DATA_BLOCK "PilzData"
VAR
  "85A1" : STRUCT
    I8 : Bool;
    I9 : Bool;
    I10 : Bool;
    I11 : Bool;
    I12 : Bool;
    I13 : Bool;
    I14 : Bool;
    I15 : Bool;
    I0 : Bool;
    I1 : Bool;
    I2 : Bool;
    I3 : Bool;
    I4 : Bool;
    I5 : Bool;
    I6 : Bool;
    I7 : Bool;
    I24 : Bool;
    I25 : Bool;
    I26 : Bool;
    I27 : Bool;
    I28 : Bool;
    I29 : Bool;
    I30 : Bool;
    I31 : Bool;
    I16 : Bool;
    I17 : Bool;
    I18 : Bool;
    I19 : Bool;
    I20 : Bool;
    I21 : Bool;
    I22 : Bool;
    I23 : Bool;
    O0 : Bool;
    O1 : Bool;
    O2 : Bool;
    O3 : Bool;
    Spare_1 : Bool;
    Spare_2 : Bool;
    Spare_3 : Bool;
    Spare_4 : Bool;
    Spare_5 : Bool;
    Spare_6 : Bool;
    Spare_7 : Bool;
    Spare_8 : Bool;
    Spare_9 : Bool;
    Spare_10 : Bool;
    Spare_11 : Bool;
    Spare_12 : Bool;
  END_STRUCT;
  "85A2" : STRUCT
    I0 : Bool;
    I1 : Bool;
    I2 : Bool;
    I3 : Bool;
    I4 : Bool;
    I5 : Bool;
    I6 : Bool;
    I7 : Bool;
    O0 : Bool;
    O1 : Bool;
    O2 : Bool;
    O3 : Bool;
    Spare_1 : Bool;
    Spare_2 : Bool;
    Spare_3 : Bool;
    Spare_4 : Bool;
  END_STRUCT;
  "85A3" : STRUCT
    I0 : Bool;
    I1 : Bool;
    I2 : Bool;
    I3 : Bool;
    I4 : Bool;
    I5 : Bool;
    I6 : Bool;
    I7 : Bool;
    O0 : Bool;
    O1 : Bool;
    O2 : Bool;
    O3 : Bool;
    Spare_1 : Bool;
    Spare_2 : Bool;
    Spare_3 : Bool;
    Spare_4 : Bool;
  END_STRUCT;
  "85A4" : STRUCT
    I0 : Bool;
    I1 : Bool;
    I2 : Bool;
    I3 : Bool;
    I4 : Bool;
    I5 : Bool;
    I6 : Bool;
    I7 : Bool;
    O0 : Bool;
    O1 : Bool;
    O2 : Bool;
    O3 : Bool;
    Spare_1 : Bool;
    Spare_2 : Bool;
    Spare_3 : Bool;
    Spare_4 : Bool;
  END_STRUCT;
  "85A5" : STRUCT
    I0 : Bool;
    I1 : Bool;
    I2 : Bool;
    I3 : Bool;
    I4 : Bool;
    I5 : Bool;
    I6 : Bool;
    I7 : Bool;
    O0 : Bool;
    O1 : Bool;
    O2 : Bool;
    O3 : Bool;
    Spare_1 : Bool;
    Spare_2 : Bool;
    Spare_3 : Bool;
    Spare_4 : Bool;
  END_STRUCT;
  TON : Array[0..50] of TON_TIME;
  OK_BoxFlag : STRUCT
    X_Moving : Bool;
    Y_Pulling : Bool;
    X_Need_MoveBox : Bool;
    Y_Need_PullBox : Bool;
    Pushing : Bool;
    ChangeUnloadingBox : Bool;
    HMIChangeUnloadingBox : Bool;
    ManualOKBox : Bool;
    HMIManualOKBox : Int;
  END_STRUCT;
  Status : Int;
END_VAR
BEGIN
END_DATA_BLOCK
